TYPE "FCP_OUT"
VERSION : 0.1
// Block: FCP_OUT
   STRUCT
      EFCControlWord : EFC_CONTROL_WORD;
      FcPControlWord : FCP_CONTROL_WORD;
      PressureCmd : Word;
      FlowCmd : Word;
   END_STRUCT;

END_TYPE
